// TIA Portal V20 export
DATA_BLOCK "ControlNodes"   // DB117
// stored: MemoryReserve 100, Namespace Unit1.Em12
   VAR
      em : "LAF_typeEmControlNode";
      emstate { S7_SetPoint := 'True'} : "LUC_typeStates";
      cm : "Unit1.Em12.typeCmControlNode";
      citiMap : Struct
         PMC : "LER_PMC_Input_Data";
         FlexNet { S7_SetPoint := 'True'} : "LER_FlexNet_Data";
      END_STRUCT;
      stackNgBox : "Unit1.Em12.typeSequenceControlNode";
      SpecialFunctionMode : Struct
         DryRun : Struct
            JRdetectPV : Array[0..15] of Bool;
         END_STRUCT;
      END_STRUCT;
      cmStackNgBoxDetect : "LBC_typeDigitalSignalControlNode";
      cmStackNgBoxFullDetect : "LBC_typeDigitalSignalControlNode";
      cmStackNgBoxLoadingUpDown : "LBC_typeTwoWayActuatorControlNode";
      cmStackNgBoxUnitMoverBwdFwd : "LBC_typeTwoWayActuatorControlNode";
      cmStackNgBoxClampLeftOpenClose : "LBC_typeTwoWayActuatorControlNode";
      cmStackNgBoxClampRightOpenClose : "LBC_typeTwoWayActuatorControlNode";
      cmStackNgBoxClampMoverOpenClose : "LBC_typeTwoWayActuatorControlNode";
      cmStackNgBoxLiftDownUp : "LBC_typeTwoWayActuatorControlNode";
      cmStackNgBoxLockDownUp : "LBC_typeTwoWayActuatorControlNode";
   END_VAR
BEGIN
END_DATA_BLOCK
